TYPE ZDataRecipe :
STRUCT
  RecipeParam1 : LREAL;
  RecipeParam2 : LREAL;
  RecipeParam3 : LREAL;
END_STRUCT
END_TYPE

(* stored: Version 1.1.0.1
   DUT ZDataRecipe: Id {bbea6db5-069b-46ef-9d05-0f841a82432d} *)
